KUKA KRL program: hp042.src, hp042.dat

--- hp042.src ---
&ACCESS RVP
&REL 4
&COMMENT Axor ETB
&PARAM DISKPATH = KRC:\R1\Program
&PARAM TEMPLATE = C:\KRC\Roboter\Template\vorgabe
&PARAM EDITMASK = *
DEF hp042( )
;FOLD INI
  ;FOLD BASISTECH INI
    GLOBAL INTERRUPT DECL 3 WHEN $STOPMESS==TRUE DO IR_STOPM ( )
    INTERRUPT ON 3
    BAS (#INITMOV,0)
  ;ENDFOLD (BASISTECH INI)
;FOLD GRIPPERTECH INI
USER_GRP(0,DUMMY,DUMMY,GDEFAULT)
;ENDFOLD (GRIPPERTECH INI)
  ;FOLD USER INI
    ;Make your modifications here

  ;ENDFOLD (USER INI)
     ;FOLD COLLISION_V_3.01 INI ;%{E}
        IF (COLLISION_DATA[1].I_NR>0) THEN
          GLOBAL INTERRUPT DECL 21 WHEN $IN[COLLISION_DATA[1].I_NR]==FALSE DO COLLSTOP (1,0 )
        ENDIF
        IF (COLLISION_DATA[2].I_NR>0) THEN
          GLOBAL INTERRUPT DECL 22 WHEN $IN[COLLISION_DATA[2].I_NR]==FALSE DO COLLSTOP (2,0 )
        ENDIF
        IF (COLLISION_DATA[3].I_NR>0) THEN
          GLOBAL INTERRUPT DECL 23 WHEN $IN[COLLISION_DATA[3].I_NR]==FALSE DO COLLSTOP (3,0 )
        ENDIF
        IF (COLLISION_DATA[4].I_NR>0) THEN
          GLOBAL INTERRUPT DECL 24 WHEN $IN[COLLISION_DATA[4].I_NR]==FALSE DO COLLSTOP (4,0 )
        ENDIF
     ;ENDFOLD (COLLISION)
;ENDFOLD (INI)

; Caracterizacao dos meios de producao
; Changes: HP042 - Axor ETB
; Versao Atual: 28/03/2016
; Name: P13.050-R4

chk_w8_wechs_ok ( )       ; CHECK TOOL CHANGE

MBINI( )                  ; RESET SINAIS

$TIMER[9]=0
$TIMER_STOP[9]=FALSE

;FOLD PTP HOME  Vel=100 % DEFAULT;%{PE}%MKUKATPBASIS,%CMOVE,%VPTP,%P 1:PTP, 2:HOME, 3:, 5:100, 7:DEFAULT
$BWDSTART = FALSE
PDAT_ACT=PDEFAULT
FDAT_ACT=FHOME
BAS(#PTP_PARAMS,100)
$H_POS=XHOME
PTP XHOME
;ENDFOLD

WKZ6_AN ( )               ; PEGA GRIPPER

HO_COM_01_ST04_G01 ( )    ; PEGA PAINEL FRONTAL

AB_COM_01_ST01_G01_OT ( )    ; DEPOSITA NA GEOBOX

WKZ5_AN ( )               ; PEGA GUN C3

PS_B_ETB_GEO_C03 ( )      ; SOLDA GEOMETRIA

WKZ5_AB ( )               ; DEPOSITA GUN C3

WKZ6_OFF_ST600 ( )        ; PEGA GRIPPER GEOBOX

WKZ6_AB ( )               ; DEPOSITA GRIPPER

WKZ5_AUX_C03 ( )          ; TRAJETORIA AUX C3

WKZ5_AN ( )               ; PEGA GUN C3

PS_B_ETB_RES_C03 ( )      ; SOLDA RESPOT

WKZ5_AB ( )               ; DEPOSITA GUN C3

;FOLD PTP HOME  Vel=100 % DEFAULT;%{PE}%MKUKATPBASIS,%CMOVE,%VPTP,%P 1:PTP, 2:HOME, 3:, 5:100, 7:DEFAULT
$BWDSTART = FALSE
PDAT_ACT=PDEFAULT
FDAT_ACT=FHOME
BAS(#PTP_PARAMS,100)
$H_POS=XHOME
PTP XHOME
;ENDFOLD

$TIMER_STOP[9]=TRUE

END

--- hp042.dat ---
&ACCESS RVP
&REL 4
&COMMENT Axor ETB
&PARAM DISKPATH = KRC:\R1\Program
&PARAM TEMPLATE = C:\KRC\Roboter\Template\vorgabe
&PARAM EDITMASK = *
DEFDAT hp042
;FOLD EXTERNAL DECLARATIONS;%{PE}%MKUKATPBASIS,%CEXT,%VCOMMON,%P
;FOLD GRIPPERTECH EXT
EXT  H50 (INT  :IN,INT  :IN,INT  :IN,GRP_TYP  :IN )
;ENDFOLD (GRIPPERTECH EXT)
;FOLD SPOTTECH EXT
EXT  USERSPOT (S_COMMAND  :IN,SPOT_TYPE  :IN )
;ENDFOLD (SPOTTECH EXT)
;FOLD BASISTECH EXT;%{PE}%MKUKATPBASIS,%CEXT,%VEXT,%P
EXT  BAS (BAS_COMMAND  :IN,REAL  :IN )
DECL INT SUCCESS
;ENDFOLD (BASISTECH EXT)
;FOLD USER EXT;%{E}%MKUKATPUSER,%CEXT,%VEXT,%P
;Make your modifications here

;ENDFOLD (USER EXT)
;ENDFOLD (EXTERNAL DECLARATIONS)
ENDDAT
